// TwinCAT 3 PLC project Reaktoreinheit_V1
// ProgramVersion: 3.1.4024.0
// libraries:
//   Tc2_Standard, * (Beckhoff Automation GmbH)
//   Tc2_System, * (Beckhoff Automation GmbH)
//   Tc2_Utilities, * (Beckhoff Automation GmbH)
//   Tc3_Module, * (Beckhoff Automation GmbH)
//   VisuDialogs, * (System)
//   VisuSymbols,3.5.10.0,System
// project tree:
//   DUTs/ I_HKSystem.TcIO, I_Magnetventil.TcIO, I_Motor1R.TcIO, I_Motor2R.TcIO (not stored), I_Sensor.TcIO (not stored), RezeptControlWord.TcDUT
//   / GlobalTextList.TcGTLO, PlcTask.TcTTO, Visualisierungsmanager.TcVMO (not stored), VISU_TASK.TcTTO (not stored)
//   GVLs/ GVL.TcGVL
//   POUs/01_Funktionblöcke/ FB_Modus.TcPOU
//   POUs/01_Funktionblöcke/01_Grundbausteine/ FB_A_HKSystem.TcPOU, FB_A_Magnetventil.TcPOU, FB_A_Motor1R.TcPOU, FB_A_Motor2R.TcPOU (not stored), FB_S_Sensor.TcPOU
//   POUs/02_Reaktoranlage/ Reaktoranlage.TcPOU
//   POUs/03_Grundfunktionen/01_Hilsbausteine/ FB_Basisfunktionalitaeten.TcPOU
//   POUs/03_Grundfunktionen/02_Grundfunktionen/ GF_Entleeren.TcPOU, GF_Halten.TcPOU, GF_Pumpen.TcPOU, GF_Ruehren.TcPOU, GF_Warten.TcPOU
//   POUs/03_Grundfunktionen/ Test.TcPOU, Zuweisung.TcPOU
//   POUs/ MAIN.TcPOU
//   VISUs/ Aktoren.TcVIS
// real-time tasks:
//   TASK PlcTask: cycle T#10ms, priority 20, ADS port 350
//   TASK VISU_TASK: cycle T#200000us, priority 30, ADS port 351

CONFIGURATION Reaktoreinheit_V1
    RESOURCE PLC ON TwinCAT3
        TASK PlcTask(INTERVAL := T#10ms, PRIORITY := 20);
        PROGRAM MAIN WITH PlcTask : MAIN;
    END_RESOURCE
END_CONFIGURATION

// ---- DUTs/RezeptControlWord.TcDUT
TYPE RezeptControlWord :
STRUCT
	CW0 	:INT;
	CW1 	:REAL;
	CW2 	:TIME;
	CW3 	:REAL;
	CW4 	:REAL;
	CW5 	:TIME;
	CW6 	:TIME;
END_STRUCT
END_TYPE

// ---- GVLs/GVL.TcGVL
{attribute 'qualified_only'}
VAR_GLOBAL
	VIS_SysReset		:BOOL;
END_VAR

// ---- DUTs/I_HKSystem.TcIO
INTERFACE I_HKSystem

END_INTERFACE

// ---- DUTs/I_Magnetventil.TcIO
INTERFACE I_Magnetventil

METHOD M_A_OEFFNEN : BOOL
VAR_INPUT
END_VAR
END_METHOD

METHOD M_A_SCHLIESSEN : BOOL
VAR_INPUT
END_VAR
END_METHOD

METHOD M_M_OEFFNEN : BOOL
VAR_INPUT
END_VAR
END_METHOD

METHOD M_M_SCHLIESSEN : BOOL
VAR_INPUT
END_VAR
END_METHOD

PROPERTY P_Status : INT
GET
END_GET
END_PROPERTY

END_INTERFACE

// ---- DUTs/I_Motor1R.TcIO
INTERFACE I_Motor1R

METHOD M_A_AN : BOOL
VAR_INPUT
END_VAR
END_METHOD

METHOD M_A_AUS : BOOL
VAR_INPUT
END_VAR
END_METHOD

METHOD M_A_START : BOOL
VAR_INPUT
END_VAR
END_METHOD

METHOD M_A_STOP : BOOL
VAR_INPUT
END_VAR
END_METHOD

METHOD M_M_AN : BOOL
VAR_INPUT
END_VAR
END_METHOD

METHOD M_M_AUS : BOOL
VAR_INPUT
END_VAR
END_METHOD

METHOD M_M_START : BOOL
VAR_INPUT
END_VAR
END_METHOD

METHOD M_M_STOP : BOOL
VAR_INPUT
END_VAR
END_METHOD

PROPERTY P_Laufzeit : TIME
GET
END_GET
END_PROPERTY

PROPERTY P_MaxDrz : INT
SET
END_SET
END_PROPERTY

PROPERTY P_Status : INT
GET
END_GET
END_PROPERTY

END_INTERFACE

// ---- POUs/MAIN.TcPOU
PROGRAM MAIN
VAR
	
	// Definieren der Prozessparameter
	Param_Menge_Entleeren			:REAL := 10;
	Param_Wartedauer				:TIME := T#10S;
	Param_Haltedauer				:TIME := T#10S;
	Param_Ruehradauer				:TIME := T#10S;
	Param_Ruehrgeschw				:REAL := 10;

	// Instanzierung der Grundfunktionen
	Entleeren		:GF_Entleeren;
	
	CW	:RezeptControlWord;
	
	
END_VAR

Reaktoranlage();
Zuweisung();
Test();

Entleeren.M_START();

CW.CW0 := 4;

END_PROGRAM

// ---- POUs/03_Grundfunktionen/02_Grundfunktionen/GF_Entleeren.TcPOU
FUNCTION_BLOCK GF_Entleeren	EXTENDS FB_Basisfunktionalitaeten
VAR_INPUT
	// Instanzieren von Sensoren mit Interfaces
	Level		:I_Sensor;
	// Instanzieren von Aktoren mit Interfaces
	Ventil		:I_Magnetventil;
	
	// Frage:
	// Wie wird aumgesetzt, dass der Inhalt in ein bestimmten Reaktor läuft
END_VAR
VAR_OUTPUT
	
END_VAR
VAR
	
END_VAR

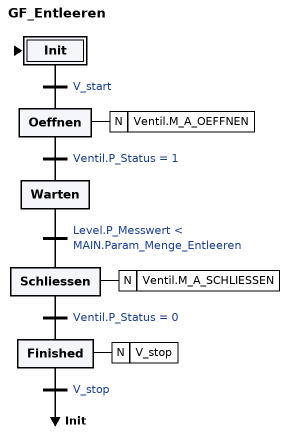
INITIAL_STEP Init:
END_STEP
TRANSITION FROM Init TO Oeffnen
    := V_start;
END_TRANSITION
STEP Oeffnen:
    Ventil.M_A_OEFFNEN(N);
END_STEP
TRANSITION FROM Oeffnen TO Warten
    := Ventil.P_Status = 1;
END_TRANSITION
STEP Warten:
END_STEP
TRANSITION FROM Warten TO Schliessen
    := Level.P_Messwert < MAIN.Param_Menge_Entleeren;
END_TRANSITION
STEP Schliessen:
    Ventil.M_A_SCHLIESSEN(N);
END_STEP
TRANSITION FROM Schliessen TO Finished
    := Ventil.P_Status = 0;
END_TRANSITION
STEP Finished:
    V_stop(N);
END_STEP
TRANSITION FROM Finished TO Init
    := V_stop;
END_TRANSITION

END_FUNCTION_BLOCK

// ---- POUs/03_Grundfunktionen/01_Hilsbausteine/FB_Basisfunktionalitaeten.TcPOU
FUNCTION_BLOCK FB_Basisfunktionalitaeten
VAR_INPUT
END_VAR
VAR_OUTPUT
END_VAR
VAR
	V_Start			:BOOL;		// Variable für internes handling der Eigenschaft 
	V_Stop			:BOOL;		// Variable für internes handling der Eigenschaft 
END_VAR

METHOD M_START : BOOL
VAR_INPUT
END_VAR
V_Start := 1;
V_Stop := 0;
END_METHOD

METHOD M_STOP : BOOL
VAR_INPUT
END_VAR
V_Start := 0;
V_Stop := 1;
END_METHOD

PROPERTY P_Ready : BOOL
GET
P_Ready := V_Stop;
END_GET
END_PROPERTY

END_FUNCTION_BLOCK

// ---- POUs/02_Reaktoranlage/Reaktoranlage.TcPOU
PROGRAM Reaktoranlage
VAR
	
	MODUS			:FB_Modus;
	
	VENTIL			:FB_A_Magnetventil; 
	RUEHRER			:FB_A_Motor1R;
	PUMPE			:FB_A_Motor2R;
	HKSYSTEM		:FB_A_HKSystem;
	
	FUELLSEN		:FB_S_Sensor;
	TEMPSEN			:FB_S_Sensor; 
	

	
END_VAR

MODUS(); // FB_Modus
VENTIL(I_iModus := MODUS.O_iModus); // FB_A_Magnetventil
FUELLSEN(); // FB_S_Sensor
RUEHRER(I_iModus := MODUS.O_iModus, I_bReset := GVL.VIS_SysReset); // FB_A_Motor1R
TEMPSEN(); // FB_S_Sensor
PUMPE(I_iModus := MODUS.O_iModus, I_bReset := GVL.VIS_SysReset); // FB_A_Motor2R
HKSYSTEM(I_iModus := MODUS.O_iModus, I_bReset := GVL.VIS_SysReset); // FB_A_HKSystem

END_PROGRAM

// ---- POUs/01_Funktionblöcke/FB_Modus.TcPOU
FUNCTION_BLOCK FB_Modus
VAR_INPUT
	I_bPower		:BOOL;
	I_bMode			:BOOL;
END_VAR

VAR_OUTPUT
	O_iModus		:INT;
	O_bMAN			:BOOL;
	O_bAUTO			:BOOL;
END_VAR

VAR
	ErrorHandling 	:SR;
END_VAR

// Handling des Betriebsmodi
IF I_bPower	THEN
	IF I_bMode THEN
		O_iModus := 1;
		O_bAUTO := FALSE;
		O_bMAN := TRUE;
	ELSE 
		O_iModus := 2;
		O_bMAN := FALSE;
		O_bAUTO := TRUE;
	END_IF
	
ELSE 
	O_iModus := 0;
	O_bMAN := FALSE;
	O_bAUTO := FALSE;
END_IF

END_FUNCTION_BLOCK

// ---- POUs/01_Funktionblöcke/01_Grundbausteine/FB_A_Magnetventil.TcPOU
FUNCTION_BLOCK FB_A_Magnetventil IMPLEMENTS I_Magnetventil
VAR_INPUT
	I_iModus			:INT;		// Zustand des Systems (z.B. 0 = AUS | 1 = MAN | 2 = AUTO)
	I_bVerriegeln		:BOOL;		// Verriegelte Elemente sind nicht ansteuerbar
END_VAR

VAR_OUTPUT
	O_bAktivieren		:BOOL;		// Ventil wird geöffnet / geschlossen
	O_bStoerung			:BOOL;		// Befindet sich das Element in einem Error
	O_iStoerungID		:INT;		// Anzeigen von Störung über eine INT-Variable
END_VAR

VAR
END_VAR

// Verriegeln des Systems (Element geht in definierten Zustand) -> Ventil wird geschlossen
IF I_bVerriegeln THEN
	O_bAktivieren := FALSE;
END_IF

METHOD M_A_OEFFNEN : BOOL
VAR_INPUT
END_VAR
// EBENE 1: Verriegelung
IF NOT I_bVerriegeln THEN	
	// EBEN 2: AUTO-Modus
		IF I_iModus = 2 THEN
			O_bAktivieren := TRUE;
		END_IF
END_IF

M_A_OEFFNEN := O_bAktivieren;
END_METHOD

METHOD M_A_SCHLIESSEN : BOOL
VAR_INPUT
END_VAR
IF I_iModus = 2 THEN
	O_bAktivieren := FALSE;
END_IF

M_A_SCHLIESSEN := NOT O_bAktivieren;
END_METHOD

METHOD M_M_OEFFNEN : BOOL
VAR_INPUT
END_VAR
// EBENE 1: Verriegelung
IF NOT I_bVerriegeln THEN	
	// EBEN 2: MAN-Modus
		IF I_iModus = 1 THEN
			O_bAktivieren := TRUE;
		END_IF
END_IF

M_M_OEFFNEN := O_bAktivieren;
END_METHOD

METHOD M_M_SCHLIESSEN : BOOL
VAR_INPUT
END_VAR
IF I_iModus = 1 THEN
	O_bAktivieren := FALSE;
END_IF

M_M_SCHLIESSEN := NOT O_bAktivieren;
END_METHOD

PROPERTY P_Status : INT
GET
IF O_bAktivieren THEN
	P_Status := 1;
ELSE
	P_Status := 0;
END_IF
END_GET
END_PROPERTY

END_FUNCTION_BLOCK

// ---- POUs/01_Funktionblöcke/01_Grundbausteine/FB_A_Motor1R.TcPOU
FUNCTION_BLOCK FB_A_Motor1R IMPLEMENTS I_Motor1R
VAR_INPUT
	I_iModus			:INT;		// Zustand des Systems (z.B. 0 = AUS | 1 = MAN | 2 = AUTO | 3 = Error)
	I_bVerriegeln		:BOOL;		// Verriegelte Elemente sind nicht ansteuerbar
	I_bReset			:BOOL;		// Zustand des Baustein wird zurückgesetzt 
	I_iGeschw			:INT;		// Angabe über Soll-Geschwindigkeit
END_VAR

VAR_OUTPUT
	O_bPower			:BOOL;		// Relais wird geschalten um FU mit Spannung zu versorgen
	O_iDrz				:INT;		// Ausgabe der Drehzahl für den Motor (Umrechnen von Spannung zu Drz)
	O_bStoerung			:BOOL;		// Befindet sich das Element in einem Error
	O_iStoerungID		:INT;		// Anzeigen von Störung über eine INT-Variable
END_VAR

VAR
	V_DrzMax		:INT;		// Variable für internes handling der Eigenschaft 
	V_Zeit			:TIME;		// Variable für internes handling der Eigenschaft 
	V_Status		:INT;		// Variable für internes handling der Eigenschaft 
	
	V_Timer			:TON;		// Runtime des Bausteins ermitteln
	
END_VAR

// Setzen der internen Variablen
P_MaxDrz := V_DrzMax;
V_Zeit := P_Laufzeit;
V_Status := P_Status;

// Reset des Bausteins
IF I_bReset THEN
	O_bStoerung := FALSE;
	O_iStoerungID := 0;
END_IF

// Verriegeln des Systems (Element geht in definierten Zustand) -> Motor wird gestoppt und ausgeschalten
IF I_bVerriegeln THEN
	O_iDrz := 0;
	O_bPower := FALSE;
END_IF

METHOD M_A_AN : BOOL
VAR_INPUT
END_VAR
// EBENE 1: Verriegelung
IF NOT I_bVerriegeln THEN	
	// EBEN 2: AUTO-Modus
		IF I_iModus = 2 THEN
			O_bPower := TRUE;
		END_IF
ELSE 
	O_bPower := FALSE;
END_IF

M_A_AN := O_bPower;
END_METHOD

METHOD M_A_AUS : BOOL
VAR_INPUT
END_VAR
IF I_iModus = 2 THEN
	O_bPower := FALSE;
	O_iDrz := 0;
END_IF

M_A_AUS := NOT O_bPower;
END_METHOD

METHOD M_A_START : BOOL
VAR_INPUT
END_VAR
// EBENE 1: Verriegelung
IF NOT I_bVerriegeln THEN

	// EBENE 2: Check der Drehzzahl
	IF I_iGeschw <= V_DrzMax THEN
		
		// Ebene 3: AUTO-Modus
		IF I_iModus = 2 THEN
			
			// EBENE 4: System muss AN sein
			IF O_bPower THEN
				O_iDrz := I_iGeschw;
				
			ELSE 	// Error: System ist nicht eingeschalten
				O_bStoerung := 1;
				O_iStoerungID := 11; 
		END_IF
		
	ELSE	// Error: Geschwindigkeit überschreitet die MaxDrz
		O_bStoerung := 1;
		O_iStoerungID := 12;
		END_IF		
	END_IF
END_IF

IF O_iDrz = I_iGeschw THEN
	M_A_START := TRUE;
ELSE
	M_A_START := FALSE;
END_IF
END_METHOD

METHOD M_A_STOP : BOOL
VAR_INPUT
END_VAR
// EBENE 1: Verriegelung
IF NOT I_bVerriegeln THEN
	O_iDrz := 0;
END_IF

IF O_iDrz = 0 THEN
	M_A_STOP := TRUE;
ELSE
	M_A_STOP := FALSE;
END_IF
END_METHOD

METHOD M_M_AN : BOOL
VAR_INPUT
END_VAR
// EBENE 1: Verriegelung
IF NOT I_bVerriegeln THEN	
	// EBEN 2: MAN-Modus
		IF I_iModus = 1 THEN
			O_bPower := TRUE;
		END_IF
ELSE 
	O_bPower := FALSE;
END_IF

M_M_AN := O_bPower;
END_METHOD

METHOD M_M_AUS : BOOL
VAR_INPUT
END_VAR
IF I_iModus = 1 THEN
	O_bPower := FALSE;
	O_iDrz := 0;
END_IF

M_M_AUS := NOT O_bPower;
END_METHOD

METHOD M_M_START : BOOL
VAR_INPUT
END_VAR
// EBENE 1: Verriegelung
IF NOT I_bVerriegeln THEN

	// EBENE 2: Check der Drehzzahl
	IF I_iGeschw <= V_DrzMax THEN
		
		// EBENE 3: MAN-Modus
		IF I_iModus = 1 THEN
			
			// EBENE 4: System muss AN sein
			IF O_bPower THEN
				O_iDrz := I_iGeschw;
				
			ELSE 	// Error: System ist nicht eingeschalten
				O_bStoerung := 1;
			O_iStoerungID := 11;
			END_IF
		END_IF
		
	ELSE	// Error: Geschwindigkeit überschreitet die MaxDrz
		O_bStoerung := 1;
		O_iStoerungID := 12;
	END_IF		
END_IF

IF O_iDrz = I_iGeschw THEN
	M_M_START := TRUE;
ELSE
	M_M_START := FALSE;
END_IF
END_METHOD

METHOD M_M_STOP : BOOL
VAR_INPUT
END_VAR
// EBENE 1: Verriegelung
IF NOT I_bVerriegeln THEN
	O_iDrz := 0;
END_IF

IF O_iDrz = 0 THEN
	M_M_STOP := TRUE;
ELSE
	M_M_STOP := FALSE;
END_IF
END_METHOD

PROPERTY PUBLIC P_Laufzeit : TIME
GET
IF O_iDrz > 0 THEN
	V_Timer(IN := TRUE, PT := T#100H);
END_IF

IF O_iDrz = 0 THEN
	V_Timer(IN := FALSE);
END_IF 
P_Laufzeit := V_Timer.ET;
END_GET
END_PROPERTY

PROPERTY PUBLIC P_MaxDrz : INT
SET
END_SET
END_PROPERTY

PROPERTY PUBLIC P_Status : INT
GET
IF O_bPower THEN
	P_Status := 1;
ELSE
	P_Status := 0;
END_IF

IF O_iDrz > 0 AND O_bPower THEN
	P_Status := 2;
ELSE
	P_Status := 1;
END_IF
END_GET
END_PROPERTY

END_FUNCTION_BLOCK

// ---- POUs/01_Funktionblöcke/01_Grundbausteine/FB_A_HKSystem.TcPOU
FUNCTION_BLOCK FB_A_HKSystem IMPLEMENTS I_HKSystem
VAR_INPUT
	I_bVerbunden	:BOOL;		// Angabe ob HK-System angeschlossen ist
	I_iModus		:INT;		// Zustand des Systems (z.B. 0 = AUS | 1 = MAN | 2 = AUTO)
	I_iTemp			:INT;		// Aktuelle Temperatur um Heizmodus auszuwählen und zu stoppen
	I_bVerriegeln	:BOOL;		// Verriegelte Elemente sind nicht ansteuerbar
	I_bReset		:BOOL;		// Zustand des Baustein wird zurückgesetzt 
END_VAR

VAR_OUTPUT
	O_bPumpen		:BOOL;		// Pumpe des HK-Systems wird betrieben
	O_bKuehlen		:BOOL;		// HK-System heizt das Medium auf
	O_bHeizen		:BOOL;		// HK-System kühlt das Medium ab
	O_bStoerung		:BOOL;		// Befindet sich das Element in einem Error
	O_iStoerungID	:INT;		// Anzeigen von Störung über eine INT-Variable
	
END_VAR
	
VAR
	V_DefTemp		:INT;		// Variable für internes handling der Eigenschaft 
	V_Zeit			:TIME;		// Variable für internes handling der Eigenschaft 
	V_Zustand		:INT;		// Variable für internes handling der Eigenschaft 
	
	V_Timer			:TON;		// Runtime des Bausteins ermitteln
END_VAR

// Setzen der internen Variablen
V_Zeit := P_Laufzeit;
V_Zustand := P_Zustand;

// Fehler durch Verbindungsabbruch
IF O_bPumpen OR O_bKuehlen OR O_bHeizen THEN
	IF NOT I_bVerbunden THEN
		O_bPumpen := FALSE;
		O_bKuehlen := FALSE;
		O_bHeizen := FALSE;
		
		O_bStoerung := TRUE;
		O_iStoerungID := 04;
	END_IF
END_IF

// Abbruch des Heiz-Kühlprozesses beim erreichen der Temp
IF O_bHeizen OR O_bKuehlen THEN 
	IF I_iTemp = V_DefTemp THEN
		O_bKuehlen := FALSE;
		O_bHeizen := FALSE;		
	END_IF
END_IF

// Reset des Bausteins
IF I_bReset THEN
	O_bStoerung := FALSE;
	O_iStoerungID := 0;
END_IF

METHOD M_A_HK_AN : BOOL
VAR_INPUT
END_VAR
// EBENE 1: Verriegelung
IF NOT I_bVerriegeln THEN	
	// EBENE 2: AUTO-Modus
		IF I_iModus = 2 THEN
			// EBENE 3: Ist Pumpe AN
				IF O_bPumpen THEN
				// EBENE 4: Heizen oder Kühlen
					IF V_DefTemp > I_iTemp THEN
						O_bKuehlen := FALSE;
						O_bHeizen := TRUE;
						
						M_A_HK_AN := O_bHeizen;
						
					ELSIF I_iTemp > V_DefTemp THEN 	
						O_bHeizen := FALSE;
						O_bKuehlen := TRUE;
						
						M_A_HK_AN := O_bKuehlen;
					END_IF
				ELSE // Error: System ist nicht eingeschalten
					O_bStoerung := 1;
					O_iStoerungID := 11; 
				END_IF
			END_IF
END_IF
END_METHOD

METHOD M_A_HK_AUS : BOOL
VAR_INPUT
END_VAR
// EBENE 1: Verriegelung
IF NOT I_bVerriegeln THEN
		O_bKuehlen := FALSE;
		O_bHeizen := FALSE;
END_IF

IF O_bKuehlen = FALSE THEN
	M_A_HK_AUS := TRUE;
END_IF
END_METHOD

METHOD M_A_PUMPE_AN : BOOL
VAR_INPUT
END_VAR
// EBENE 1: Verriegelung
IF NOT I_bVerriegeln THEN	
	// EBENE 2: AUTO-Modus
		IF I_iModus = 2 THEN
			// EBENE 3: System muss angeschlossen sein
			IF I_bVerbunden THEN
				O_bPumpen := TRUE;
			ELSE 	// Error: System ist nicht angeschlossen
				O_bStoerung := 1;
				O_iStoerungID := 03;
			END_IF
		END_IF
END_IF

M_A_PUMPE_AN := O_bPumpen;
END_METHOD

METHOD M_A_PUMPE_AUS : BOOL
VAR_INPUT
END_VAR
// EBENE 1: Verriegelung
IF NOT I_bVerriegeln THEN
	IF NOT O_bHeizen AND NOT O_bKuehlen THEN
		O_bPumpen := FALSE;
	ELSE
		O_bStoerung := TRUE;
		O_iStoerungID := 05;
	END_IF
END_IF

IF O_bPumpen = FALSE THEN
	M_A_PUMPE_AUS := TRUE;
END_IF
END_METHOD

METHOD M_M_HK_AN : BOOL
VAR_INPUT
END_VAR
// EBENE 1: Verriegelung
IF NOT I_bVerriegeln THEN	
	// EBENE 2: MAN-Modus
		IF I_iModus = 1 THEN
			// EBENE 3: Ist Pumpe AN
				IF O_bPumpen THEN
				// EBENE 4: Heizen oder Kühlen
					IF V_DefTemp > I_iTemp THEN
						O_bKuehlen := FALSE;
						O_bHeizen := TRUE;
						
						M_M_HK_AN := O_bHeizen;
						
					ELSIF I_iTemp > V_DefTemp THEN 	
						O_bHeizen := FALSE;
						O_bKuehlen := TRUE;
						
						M_M_HK_AN := O_bKuehlen;
					END_IF
				ELSE // Error: System ist nicht eingeschalten
				O_bStoerung := 1;
				O_iStoerungID := 11; 	
				END_IF
			END_IF
END_IF
END_METHOD

METHOD M_M_HK_AUS : BOOL
VAR_INPUT
END_VAR
// EBENE 1: Verriegelung
IF NOT I_bVerriegeln THEN
		O_bKuehlen := FALSE;
		O_bHeizen := FALSE;
END_IF

IF O_bKuehlen = FALSE THEN
	M_M_HK_AUS := TRUE;
END_IF
END_METHOD

METHOD M_M_PUMPE_AN : BOOL
VAR_INPUT
END_VAR
// EBENE 1: Verriegelung
IF NOT I_bVerriegeln THEN	
	// EBENE 2: MAN-Modus
		IF I_iModus = 1 THEN
			// EBENE 3: System muss angeschlossen sein
			IF I_bVerbunden THEN
				O_bPumpen := TRUE;
			ELSE 	// Error: System ist nicht angeschlossen
				O_bStoerung := 1;
				O_iStoerungID := 03;
			END_IF
		END_IF
END_IF

M_M_PUMPE_AN := O_bPumpen;
END_METHOD

METHOD M_M_PUMPE_AUS : BOOL
VAR_INPUT
END_VAR
// EBENE 1: Verriegelung
IF NOT I_bVerriegeln THEN
	IF NOT O_bHeizen AND NOT O_bKuehlen THEN
		O_bPumpen := FALSE;
	ELSE
		O_bStoerung := TRUE;
		O_iStoerungID := 05;
	END_IF
END_IF

IF O_bPumpen = FALSE THEN
	M_M_PUMPE_AUS := TRUE;
END_IF
END_METHOD

PROPERTY P_DefTemp : INT
SET
END_SET
END_PROPERTY

PROPERTY P_Laufzeit : TIME
GET
IF O_bKuehlen OR O_bHeizen THEN
	V_Timer(IN := TRUE, PT := T#100H);
ELSE
	V_Timer(IN := FALSE);
END_IF

P_Laufzeit := V_Timer.ET;
END_GET
END_PROPERTY

PROPERTY PUBLIC P_Zustand : INT
GET
END_GET
END_PROPERTY

END_FUNCTION_BLOCK

// ---- POUs/01_Funktionblöcke/01_Grundbausteine/FB_S_Sensor.TcPOU
FUNCTION_BLOCK FB_S_Sensor IMPLEMENTS	I_Sensor	
VAR_INPUT
	I_iSignal			:INT;		// Messsignal des Sensors
	I_rHigh				:REAL;		// Oberer Schwellenwert für Prozess
	I_rLow				:REAL;		// Unterer Schwellenwert für Prozess
	I_rMax				:REAL;		// Skallierungswert -> Max-Wert 
	I_rMin				:REAL;		// Skallierungswert -> Min-Wert 
END_VAR

VAR_OUTPUT
	O_bStoerung			:BOOL;		// Befindet sich das Element in einem Error
	O_iStoerungID		:INT;		// Anzeigen von Störung über eine INT-Variable
END_VAR

VAR
	Messwert			:REAL;		// Wert für HMI
	GrenzeOben			:BOOL;		// Wert für HMI
	GrenzeUnten			:BOOL;		// Wert für HMI
END_VAR

Messwert := P_Messwert;
GrenzeOben := P_GrenzeOben;
GrenzeUnten := P_GrenzeUnten;

PROPERTY PUBLIC P_GrenzeOben : BOOL
GET
IF P_Messwert > I_rHigh THEN
	P_GrenzeOben := TRUE;
ELSE
	P_GrenzeOben := FALSE;
END_IF
END_GET
END_PROPERTY

PROPERTY PUBLIC P_GrenzeUnten : BOOL
GET
IF P_Messwert < I_rLow THEN
	P_GrenzeUnten := TRUE;
ELSE
	P_GrenzeUnten := FALSE;
END_IF
END_GET
END_PROPERTY

PROPERTY PUBLIC P_Messwert : REAL
GET
IF I_iSignal > 27648 OR I_iSignal < 0 THEN
	O_bStoerung := TRUE;
	O_iStoerungID := 04;
ELSE
	O_bStoerung := FALSE; 
END_IF

// Linearisierung des Wertes 
P_Messwert := INT_TO_REAL(I_iSignal) * (I_rMax-I_rMin) / 27648 + I_rMin;
END_GET
END_PROPERTY

END_FUNCTION_BLOCK

// ---- POUs/03_Grundfunktionen/Zuweisung.TcPOU
PROGRAM Zuweisung
VAR

END_VAR

Main.Entleeren(Level := Reaktoranlage.FUELLSEN, Ventil := Reaktoranlage.VENTIL); // GF_Entleeren

END_PROGRAM

// ---- POUs/03_Grundfunktionen/Test.TcPOU
PROGRAM Test
VAR
END_VAR

IF TRUE THEN
	Act_Test();
END_IF

ACTION Act_Test:
MAIN.Entleeren(); // GF_Entleeren
END_ACTION

END_PROGRAM

// ---- POUs/03_Grundfunktionen/02_Grundfunktionen/GF_Halten.TcPOU
FUNCTION_BLOCK GF_Halten EXTENDS FB_Basisfunktionalitaeten
VAR_INPUT
	// Instanzieren von Sensoren mit Interfaces
	
	// Instanzieren von Aktoren mit Interfaces
	
END_VAR
VAR_OUTPUT
	
END_VAR
VAR
	
END_VAR

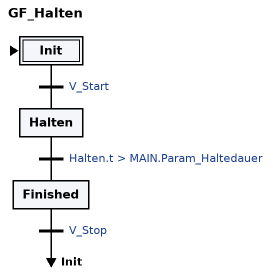
INITIAL_STEP Init:
END_STEP
TRANSITION FROM Init TO Halten
    := V_Start;
END_TRANSITION
STEP Halten:
END_STEP
TRANSITION FROM Halten TO Finished
    := Halten.t > MAIN.Param_Haltedauer;
END_TRANSITION
STEP Finished:
END_STEP
TRANSITION FROM Finished TO Init
    := V_Stop;
END_TRANSITION

END_FUNCTION_BLOCK

// ---- POUs/03_Grundfunktionen/02_Grundfunktionen/GF_Pumpen.TcPOU
FUNCTION_BLOCK GF_Pumpen EXTENDS FB_Basisfunktionalitaeten
VAR_INPUT
	// Instanzieren von Sensoren mit Interfaces
	
	// Instanzieren von Aktoren mit Interfaces
	
	
END_VAR
VAR_OUTPUT
	
END_VAR
VAR
	
END_VAR

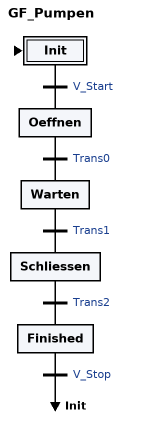
INITIAL_STEP Init:
END_STEP
TRANSITION FROM Init TO Oeffnen
    := V_Start;
END_TRANSITION
STEP Oeffnen:
END_STEP
TRANSITION FROM Oeffnen TO Warten
    := Trans0;
END_TRANSITION
STEP Warten:
END_STEP
TRANSITION FROM Warten TO Schliessen
    := Trans1;
END_TRANSITION
STEP Schliessen:
END_STEP
TRANSITION FROM Schliessen TO Finished
    := Trans2;
END_TRANSITION
STEP Finished:
END_STEP
TRANSITION FROM Finished TO Init
    := V_Stop;
END_TRANSITION

END_FUNCTION_BLOCK

// ---- POUs/03_Grundfunktionen/02_Grundfunktionen/GF_Ruehren.TcPOU
FUNCTION_BLOCK GF_Ruehren EXTENDS FB_Basisfunktionalitaeten
VAR_INPUT
	// Instanzieren von Sensoren mit Interfaces
	
	// Instanzieren von Aktoren mit Interfaces
	Ruehrer		:I_Motor1R;
	
	
	// Fragen
	// Wo definiere ich die gewschwindigkeit oder wie kommt diese zum Funktionsblock? 
	// Wird die Geschwindigkeit über den Shrittablauf definiert? 
END_VAR
VAR_OUTPUT
	
END_VAR
VAR
	
END_VAR

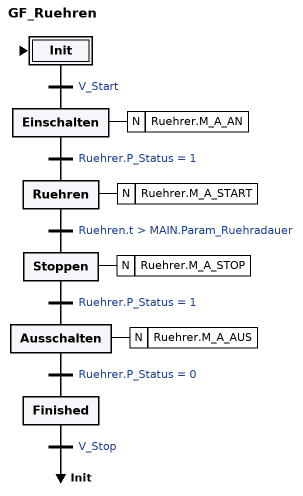
INITIAL_STEP Init:
END_STEP
TRANSITION FROM Init TO Einschalten
    := V_Start;
END_TRANSITION
STEP Einschalten:
    Ruehrer.M_A_AN(N);
END_STEP
TRANSITION FROM Einschalten TO Ruehren
    := Ruehrer.P_Status = 1;
END_TRANSITION
STEP Ruehren:
    Ruehrer.M_A_START(N);
END_STEP
TRANSITION FROM Ruehren TO Stoppen
    := Ruehren.t > MAIN.Param_Ruehradauer;
END_TRANSITION
STEP Stoppen:
    Ruehrer.M_A_STOP(N);
END_STEP
TRANSITION FROM Stoppen TO Ausschalten
    := Ruehrer.P_Status = 1;
END_TRANSITION
STEP Ausschalten:
    Ruehrer.M_A_AUS(N);
END_STEP
TRANSITION FROM Ausschalten TO Finished
    := Ruehrer.P_Status = 0;
END_TRANSITION
STEP Finished:
END_STEP
TRANSITION FROM Finished TO Init
    := V_Stop;
END_TRANSITION

END_FUNCTION_BLOCK

// ---- POUs/03_Grundfunktionen/02_Grundfunktionen/GF_Warten.TcPOU
FUNCTION_BLOCK GF_Warten EXTENDS FB_Basisfunktionalitaeten
VAR_INPUT
	// Instanzieren von Sensoren mit Interfaces
	
	// Instanzieren von Aktoren mit Interfaces
	
END_VAR
VAR_OUTPUT
	
END_VAR
VAR
	
END_VAR

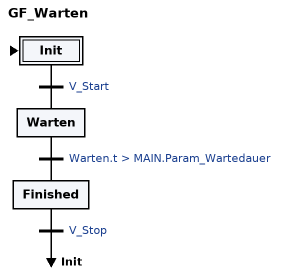
INITIAL_STEP Init:
END_STEP
TRANSITION FROM Init TO Warten
    := V_Start;
END_TRANSITION
STEP Warten:
END_STEP
TRANSITION FROM Warten TO Finished
    := Warten.t > MAIN.Param_Wartedauer;
END_TRANSITION
STEP Finished:
END_STEP
TRANSITION FROM Finished TO Init
    := V_Stop;
END_TRANSITION

END_FUNCTION_BLOCK

// ---- GlobalTextList.TcGTLO
TEXTLIST GlobalTextList
  307 = '%d'
  665 = '%i'
  57 = '%s'
  569 = '100'
  663 = 'AUTO'
  961 = 'Button'
  792 = 'd'
  881 = 'Eigenschaften'
  225 = 'FB_Füllstandsensor'
  379 = 'FB_HKSystem'
  606 = 'FB_Magnetventil'
  583 = 'FB_Motor1R'
  65 = 'FB_Motor2R'
  234 = 'FB_Temperatursensor'
  111 = 'FB_Tempoeratursensor'
  808 = 'GET'
  947 = 'Gruppenfeld'
  745 = 'Inputs'
  999 = 'I_iGeschw'
  589 = 'I_iHeizMode'
  584 = 'I_iHeizModus'
  510 = 'I_iSignal'
  254 = 'I_iTemp'
  916 = 'I_rHigh'
  121 = 'I_rLow'
  362 = 'I_rMax'
  680 = 'I_rMin'
  331 = 'Magnetventil'
  348 = 'MAN'
  64 = 'Methodenhandling'
  581 = 'MODI:'
  242 = 'Modus'
  468 = 'Modus:'
  654 = 'MODUS:'
  278 = 'M_M_AN'
  0 = 'M_M_AUS'
  843 = 'M_M_BWD'
  38 = 'M_M_FWD'
  739 = 'M_M_HK_AN'
  330 = 'M_M_HK_AUS'
  478 = 'M_M_OEFFNEN'
  994 = 'M_M_PUMPE_AN'
  78 = 'M_M_PUMPE_AUS'
  727 = 'M_M_SCHLIESSEN'
  150 = 'M_M_START'
  41 = 'M_M_STOP'
  28 = 'Outputs '
  547 = 'O_bAktivieren'
  721 = 'O_bError'
  2 = 'O_bHeizen'
  342 = 'O_bKuehlen'
  866 = 'O_bPower'
  746 = 'O_bPumpen'
  544 = 'O_bRichtung'
  418 = 'O_iDrz'
  518 = 'O_iStoerungID'
  932 = 'POWER:'
  685 = 'P_GrenzeOben'
  502 = 'P_GrenzeUnten'
  794 = 'P_Laufzeit'
  293 = 'P_MaxDrz'
  692 = 'P_Messwert'
  758 = 'P_Zustand'
  954 = 'RESET:'
  119 = 'Schliessen'
  833 = 'sd'
  332 = 'SET'
  157 = 'TBD'
  412 = 'test'
  465 = 'Test'
  901 = 'Ventil aktiviert:'
  993 = 'Verbunden'
  834 = 'VERBUNDEN:'
  152 = 'VERRIEGELN:'
  664 = 'VERRIEGELUNG'
  212 = 'VERRIEGELUNG:'
  258 = 'Öffnen'
END_TEXTLIST

// ---- VISUs/Aktoren.TcVIS
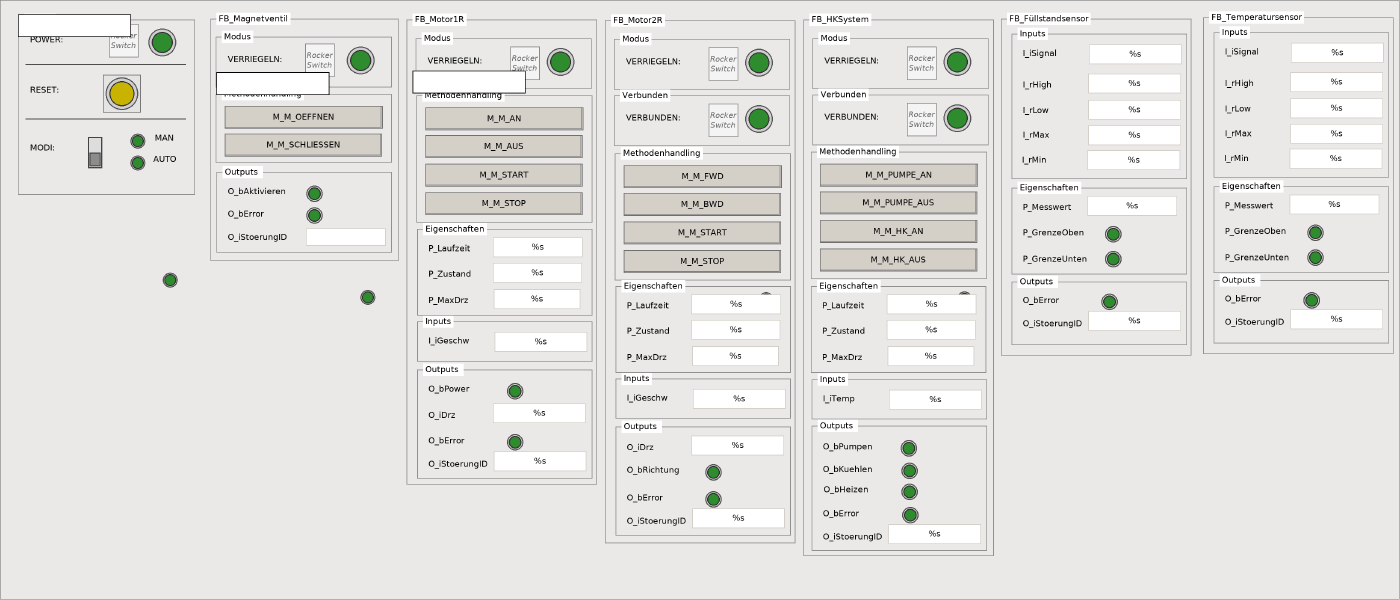
VISUALIZATION Aktoren  // 1863x799
    Rectangle (-1,-1 1863x799)
    GroupBox (280,17 250x330), "FB_Magnetventil"
        Textfield (127,287 106x23), text variable: Reaktoranlage.VENTIL.O_iStoerungID
    GroupBox (287,41 234x75), "Modus"
        Label (13,23 150x30), "VERRIEGELN:"
        Lamp1 (172,18 42x43), variable: Reaktoranlage.VENTIL.I_bVerriegeln, style: Lamp-Lamp1-Green
        Lamp1 (191,340 23x30), style: Lamp-Lamp1-Green
    RockerSwitch (406,58 39x44), variable: Reaktoranlage.VENTIL.I_bVerriegeln, behaviour: TOGGLE, style: Switch-RockerSwitch-Gray
    GroupBox (287,117 234x99), "Methodenhandling"
        Rectangle (-530,-100 150x30)
        Button (12,24 210x30), "M_M_OEFFNEN"
            OnMouseClick: execute { Reaktoranlage.VENTIL.M_M_OEFFNEN(); }
        Button (12,61 209x30), "M_M_SCHLIESSEN"
            OnMouseClick: execute { Reaktoranlage.VENTIL.M_M_SCHLIESSEN(); }
    GroupBox (288,221 233x115), "Outputs"
        Label (12,19 150x30), "O_bAktivieren"
        Label (12,49 150x30), "O_bError"
        Label (12,80 150x30), "O_iStoerungID"
        Lamp1 (118,22 25x30), variable: Reaktoranlage.VENTIL.O_bAktivieren, style: Lamp-Lamp1-Green
        Lamp1 (118,51 25x30), variable: Reaktoranlage.VENTIL.O_bStoerung, style: Lamp-Lamp1-Green
    GroupBox (24,18 235x241), "Modus"
        Label (13,20 150x30), "POWER:"
        RockerSwitch (121,14 39x44), variable: Reaktoranlage.Modus.I_bPower, behaviour: TOGGLE, style: Switch-RockerSwitch-Gray
        Label (13,164 150x30), "MODI:"
        DipSwitch (82,161 41x48), variable: Reaktoranlage.Modus.I_bMode, behaviour: TOGGLE, style: Switch-DipSwitch-Gray
        Lamp1 (148,155 23x30), variable: Reaktoranlage.Modus.O_bMAN, style: Lamp-Lamp1-Green
        Lamp1 (148,184 23x30), variable: Reaktoranlage.Modus.O_bAUTO, style: Lamp-Lamp1-Green
        Label (177,179 46x30), "AUTO"
        Lamp1 (191,340 23x30), style: Lamp-Lamp1-Green
        Line (10,67) (223,67)
        Lamp1 (171,17 42x43), variable: Reaktoranlage.Modus.I_bPower, style: Lamp-Lamp1-Green
        Label (179,151 46x30), "MAN"
        Label (13,87 150x30), "RESET:"
        PushSwitch (113,80 50x53), variable: GVL.VIS_SysReset, behaviour: TAP, style: Switch-PushSwitch-Yellow
        Line (10,140) (223,140)
    GroupBox (541,18 253x627), "FB_Motor1R"
        GroupBox (12,25 234x75), "Modus"
            Label (13,23 150x30), "VERRIEGELN:"
            Lamp1 (172,18 42x43), variable: Reaktoranlage.RUEHRER.I_bVerriegeln, style: Lamp-Lamp1-Green
            Lamp1 (191,340 23x30), style: Lamp-Lamp1-Green
            RockerSwitch (126,19 39x44), variable: Reaktoranlage.RUEHRER.I_bVerriegeln, behaviour: TOGGLE, style: Switch-RockerSwitch-Gray
        GroupBox (13,101 234x177), "Methodenhandling"
            Rectangle (-530,-100 150x30)
            Button (12,24 210x30), "M_M_AN"
                OnMouseClick: execute { Reaktoranlage.RUEHRER.M_M_AN(); }
            Button (12,61 209x30), "M_M_AUS"
                OnMouseClick: execute { Reaktoranlage.RUEHRER.M_M_AUS(); }
            Button (12,99 209x30), "M_M_START"
                OnMouseClick: execute { Reaktoranlage.RUEHRER.M_M_START(); }
            Button (12,137 209x30), "M_M_STOP"
                OnMouseClick: execute { Reaktoranlage.RUEHRER.M_M_STOP(); }
        GroupBox (14,402 233x61), "Inputs"
            Label (12,19 150x30), "I_iGeschw"
            Textfield (103,22 123x26), "%s", text variable: Reaktoranlage.RUEHRER.I_iGeschw
                OnMouseClick: write Reaktoranlage.RUEHRER.I_iGeschw via Edit, min 0
        GroupBox (14,279 233x123), "Eigenschaften"
            Label (12,19 150x30), "P_Laufzeit"
            Label (12,88 150x30), "P_MaxDrz"
            Label (12,53 150x30), "P_Zustand"
            Textfield (101,53 118x26), "%s", text variable: Reaktoranlage.RUEHRER.V_Status, input disabled if: TRUE
            Textfield (102,88 115x26), "%s", text variable: Reaktoranlage.RUEHRER.V_DrzMax
                OnMouseClick: write Reaktoranlage.RUEHRER.V_DrzMax via Default
            Textfield (101,19 119x26), "%s", text variable: Reaktoranlage.RUEHRER.V_Zeit, input disabled if: TRUE
        GroupBox (14,466 233x153), "Outputs"
            Label (12,19 150x30), "O_bPower"
            Label (12,88 150x30), "O_bError"
            Label (12,119 150x30), "O_iStoerungID"
            Lamp1 (118,22 25x30), variable: Reaktoranlage.RUEHRER.O_bPower, style: Lamp-Lamp1-Green
            Lamp1 (118,90 25x30), variable: Reaktoranlage.RUEHRER.O_bStoerung, style: Lamp-Lamp1-Green
            Textfield (101,53 123x26), "%s", text variable: Reaktoranlage.RUEHRER.O_iDrz, input disabled if: TRUE
            Textfield (102,117 123x26), "%s", text variable: Reaktoranlage.RUEHRER.O_iStoerungID, input disabled if: TRUE
            Label (12,54 150x30), "O_iDrz"
    GroupBox (805,19 253x704), "FB_Motor2R"
        GroupBox (12,25 234x75), "Modus"
            Label (13,23 150x30), "VERRIEGELN:"
            Lamp1 (172,18 42x43), variable: Reaktoranlage.PUMPE.I_bVerriegeln, style: Lamp-Lamp1-Green
            Lamp1 (191,340 23x30), style: Lamp-Lamp1-Green
            RockerSwitch (126,19 39x44), variable: Reaktoranlage.PUMPE.I_bVerriegeln, behaviour: TOGGLE, style: Switch-RockerSwitch-Gray
        GroupBox (13,177 234x177), "Methodenhandling"
            Rectangle (-530,-100 150x30)
            Button (12,24 210x30), "M_M_FWD"
                OnMouseClick: execute { Reaktoranlage.PUMPE.M_M_FWD(); }
            Button (12,61 209x30), "M_M_BWD"
                OnMouseClick: execute { Reaktoranlage.PUMPE.M_M_BWD(); }
            Button (12,99 209x30), "M_M_START"
                OnMouseClick: execute { Reaktoranlage.PUMPE.M_M_START(); }
            Button (12,137 209x30), "M_M_STOP"
                OnMouseClick: execute { Reaktoranlage.PUMPE.M_M_STOP(); }
        GroupBox (14,477 233x61), "Inputs"
            Label (12,19 150x30), "I_iGeschw"
            Textfield (103,22 123x26), "%s", text variable: Reaktoranlage.PUMPE.I_iGeschw
                OnMouseClick: write Reaktoranlage.PUMPE.I_iGeschw via Edit, min 0
        GroupBox (14,354 233x123), "Eigenschaften"
            Label (12,19 150x30), "P_Laufzeit"
            Label (12,88 150x30), "P_MaxDrz"
            Label (12,53 150x30), "P_Zustand"
            Textfield (101,53 118x26), "%s", text variable: Reaktoranlage.PUMPE.V_Zustand, input disabled if: TRUE
            Textfield (102,88 115x26), "%s", text variable: Reaktoranlage.PUMPE.V_DrzMax
                OnMouseClick: write Reaktoranlage.PUMPE.V_DrzMax via Default
            Textfield (101,19 119x26), "%s", text variable: Reaktoranlage.PUMPE.V_Zeit, input disabled if: TRUE
        GroupBox (14,541 233x153), "Outputs"
            Label (12,51 150x30), "O_bRichtung"
            Label (12,88 150x30), "O_bError"
            Label (12,119 150x30), "O_iStoerungID"
            Lamp1 (118,54 25x30), variable: Reaktoranlage.PUMPE.O_bRichtung, style: Lamp-Lamp1-Green
            Lamp1 (118,90 25x30), variable: Reaktoranlage.PUMPE.O_bStoerung, style: Lamp-Lamp1-Green
            Textfield (101,20 123x26), "%s", text variable: Reaktoranlage.PUMPE.O_iDrz, input disabled if: TRUE
            Textfield (102,117 123x26), "%s", text variable: Reaktoranlage.PUMPE.O_iStoerungID, input disabled if: TRUE
            Label (12,21 150x30), "O_iDrz"
        GroupBox (12,100 234x75), "Verbunden"
            Label (13,23 150x30), "VERBUNDEN:"
            Lamp1 (172,18 42x43), variable: Reaktoranlage.PUMPE.I_bVerbunden, style: Lamp-Lamp1-Green
            RockerSwitch (126,19 39x44), variable: Reaktoranlage.PUMPE.I_bVerbunden, behaviour: TOGGLE, style: Switch-RockerSwitch-Gray
    GroupBox (1069,18 253x722), "FB_HKSystem"
        GroupBox (12,25 234x75), "Modus"
            Label (13,23 150x30), "VERRIEGELN:"
            Lamp1 (172,18 42x43), variable: Reaktoranlage.HKSYSTEM.I_bVerriegeln, style: Lamp-Lamp1-Green
            Lamp1 (191,340 23x30), style: Lamp-Lamp1-Green
            RockerSwitch (126,19 39x44), variable: Reaktoranlage.HKSYSTEM.I_bVerriegeln, behaviour: TOGGLE, style: Switch-RockerSwitch-Gray
        GroupBox (12,100 234x75), "Verbunden"
            Label (13,23 150x30), "VERBUNDEN:"
            Lamp1 (172,18 42x43), variable: Reaktoranlage.HKSYSTEM.I_bVerbunden, style: Lamp-Lamp1-Green
            RockerSwitch (126,19 39x44), variable: Reaktoranlage.HKSYSTEM.I_bVerbunden, behaviour: TOGGLE, style: Switch-RockerSwitch-Gray
        GroupBox (10,176 234x177), "Methodenhandling"
            Rectangle (-530,-100 150x30)
            Button (12,24 210x30), "M_M_PUMPE_AN"
                OnMouseClick: execute { Reaktoranlage.HKSYSTEM.M_M_PUMPE_AN(); }
            Button (12,61 209x30), "M_M_PUMPE_AUS"
                OnMouseClick: execute { Reaktoranlage.HKSYSTEM.M_M_PUMPE_AUS(); }
            Button (12,99 209x30), "M_M_HK_AN"
                OnMouseClick: execute { Reaktoranlage.HKSYSTEM.M_M_HK_AN(); }
            Button (12,137 209x30), "M_M_HK_AUS"
                OnMouseClick: execute { Reaktoranlage.HKSYSTEM.M_M_HK_AUS(); }
        GroupBox (11,541 233x174), "Outputs"
            Label (12,51 150x30), "O_bKuehlen"
            Label (12,110 150x30), "O_bError"
            Label (12,141 150x30), "O_iStoerungID"
            Lamp1 (118,53 25x30), variable: Reaktoranlage.HKSYSTEM.O_bKuehlen, style: Lamp-Lamp1-Green
            Lamp1 (119,112 25x30), variable: Reaktoranlage.HKSYSTEM.O_bStoerung, style: Lamp-Lamp1-Green
            Textfield (102,139 123x26), "%s", text variable: Reaktoranlage.HKSYSTEM.O_iStoerungID, input disabled if: TRUE
            Label (12,21 150x30), "O_bPumpen"
            Label (13,78 150x30), "O_bHeizen"
            Lamp1 (118,81 25x30), variable: Reaktoranlage.HKSYSTEM.O_bHeizen, style: Lamp-Lamp1-Green
            Lamp1 (117,23 25x30), variable: Reaktoranlage.HKSYSTEM.O_bPumpen, style: Lamp-Lamp1-Green
        GroupBox (11,479 233x61), "Inputs"
            Label (12,19 150x30), "I_iTemp"
            Textfield (103,22 123x26), "%s", text variable: Reaktoranlage.HKSYSTEM.I_iTemp
                OnMouseClick: write Reaktoranlage.HKSYSTEM.I_iTemp via Edit, min 0
        GroupBox (10,355 233x123), "Eigenschaften"
            Label (12,19 150x30), "P_Laufzeit"
            Label (12,88 150x30), "P_MaxDrz"
            Label (12,53 150x30), "P_Zustand"
            Textfield (101,53 118x26), "%s", text variable: Reaktoranlage.HKSYSTEM.V_Zustand, input disabled if: TRUE
            Textfield (102,88 115x26), "%s", text variable: Reaktoranlage.HKSYSTEM.V_DefTemp
                OnMouseClick: write Reaktoranlage.HKSYSTEM.V_DefTemp via Default
            Textfield (101,19 119x26), "%s", text variable: Reaktoranlage.HKSYSTEM.V_Zeit, input disabled if: TRUE
    GroupBox (1332,17 253x456), "FB_Füllstandsensor"
        GroupBox (14,20 233x201), "Inputs"
            Label (12,19 150x30), "I_iSignal"
            Textfield (103,22 123x26), "%s", text variable: Reaktoranlage.FUELLSEN.I_iSignal
                OnMouseClick: write Reaktoranlage.FUELLSEN.I_iSignal via Edit, min 0
            Label (12,61 150x30), "I_rHigh"
            Label (12,95 150x30), "I_rLow"
            Label (12,128 150x30), "I_rMax"
            Label (11,161 150x30), "I_rMin"
        GroupBox (14,225 233x123), "Eigenschaften"
            Label (12,19 150x30), "P_Messwert"
            Label (12,88 150x30), "P_GrenzeUnten"
            Label (12,53 150x30), "P_GrenzeOben"
            Textfield (101,19 119x26), "%s", text variable: Reaktoranlage.FUELLSEN.Messwert, input disabled if: TRUE
            Lamp1 (123,55 25x30), variable: Reaktoranlage.FUELLSEN.GrenzeOben, style: Lamp-Lamp1-Green
            Lamp1 (123,88 25x30), variable: Reaktoranlage.FUELLSEN.GrenzeUnten, style: Lamp-Lamp1-Green
        GroupBox (14,350 233x92), "Outputs"
            Label (12,18 150x30), "O_bError"
            Label (12,49 150x30), "O_iStoerungID"
            Lamp1 (118,20 25x30), variable: Reaktoranlage.FUELLSEN.O_bStoerung, style: Lamp-Lamp1-Green
            Textfield (102,47 123x26), "%s", text variable: Reaktoranlage.PUMPE.O_iStoerungID, input disabled if: TRUE
        Textfield (116,81 123x26), "%s", text variable: Reaktoranlage.FUELLSEN.I_rHigh
            OnMouseClick: write Reaktoranlage.FUELLSEN.I_rHigh via Edit, min 0
        Textfield (116,116 123x26), "%s", text variable: Reaktoranlage.FUELLSEN.I_rMin
            OnMouseClick: write Reaktoranlage.FUELLSEN.I_rLow via Edit, min 0
        Textfield (116,150 123x26), "%s", text variable: Reaktoranlage.FUELLSEN.I_rMax
            OnMouseClick: write Reaktoranlage.FUELLSEN.I_rMax via Edit, min 0
        Textfield (115,183 123x26), "%s", text variable: Reaktoranlage.FUELLSEN.I_rMin
            OnMouseClick: write Reaktoranlage.FUELLSEN.I_rMin via Edit, min 0
    GroupBox (1601,15 253x456), "FB_Temperatursensor"
        GroupBox (14,20 233x201), "Inputs"
            Label (12,19 150x30), "I_iSignal"
            Textfield (103,22 123x26), "%s", text variable: Reaktoranlage.FUELLSEN.I_iSignal
                OnMouseClick: write Reaktoranlage.TEMPSEN.I_rMin via Edit, min 0
            Label (12,61 150x30), "I_rHigh"
            Label (12,95 150x30), "I_rLow"
            Label (12,128 150x30), "I_rMax"
            Label (11,161 150x30), "I_rMin"
        GroupBox (14,225 233x123), "Eigenschaften"
            Label (12,19 150x30), "P_Messwert"
            Label (12,88 150x30), "P_GrenzeUnten"
            Label (12,53 150x30), "P_GrenzeOben"
            Textfield (101,19 119x26), "%s", text variable: Reaktoranlage.TEMPSEN.Messwert, input disabled if: TRUE
            Lamp1 (123,55 25x30), variable: Reaktoranlage.TEMPSEN.GrenzeOben, style: Lamp-Lamp1-Green
            Lamp1 (123,88 25x30), variable: Reaktoranlage.TEMPSEN.GrenzeUnten, style: Lamp-Lamp1-Green
        GroupBox (14,350 233x92), "Outputs"
            Label (12,18 150x30), "O_bError"
            Label (12,49 150x30), "O_iStoerungID"
            Lamp1 (118,20 25x30), variable: Reaktoranlage.TEMPSEN.O_bStoerung, style: Lamp-Lamp1-Green
            Textfield (102,47 123x26), "%s", text variable: Reaktoranlage.TEMPSEN.O_iStoerungID, input disabled if: TRUE
        Textfield (116,81 123x26), "%s", text variable: Reaktoranlage.FUELLSEN.I_rHigh
            OnMouseClick: write Reaktoranlage.TEMPSEN.I_rHigh via Edit, min 0
        Textfield (116,116 123x26), "%s", text variable: Reaktoranlage.FUELLSEN.I_rMin
            OnMouseClick: write Reaktoranlage.TEMPSEN.I_rLow via Edit, min 0
        Textfield (116,150 123x26), "%s", text variable: Reaktoranlage.FUELLSEN.I_rMax
            OnMouseClick: write Reaktoranlage.TEMPSEN.I_rMax via Edit, min 0
        Textfield (115,183 123x26), "%s", text variable: Reaktoranlage.TEMPSEN.O_iStoerungID
            OnMouseClick: write Reaktoranlage.TEMPSEN.I_rMin via Edit, min 0
END_VISUALIZATION
